TYPE DUT : BOOL; END_TYPE

(* stored: Version 1.1.0.1, ProductVersion 3.1.4024.12
   DUT DUT: Id {83eac58f-dab3-4d86-8a2d-b8d75b1a9a73} *)
